TYPE E_FastenerStatus : (
    FASTENER_UNKNOWN := 0,
    FASTENER_EMPTY := 10,
    FASTENER_SINGLE_OK := 20,
    FASTENER_WRONG_TYPE := 30,
    FASTENER_MULTIPLE := 40,
    FASTENER_JAMMED := 50,
    FASTENER_FAULT := 100
); END_TYPE

(* stored: Version 1.1.0.1
   DUT E_FastenerStatus: Id {E3000000-0000-4000-8000-000000000017} *)
